Universal Robots PolyScope program: tcp_debug.urp

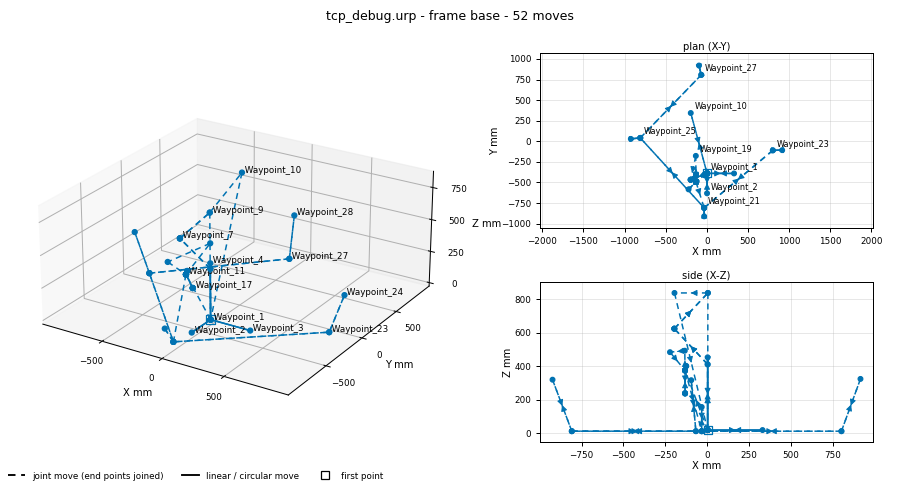
[picture p0: tool path of tcp_debug.urp in frame base, 52 of 52 moves have a stored position in this frame; points joined in program order, loops and branches not executed]
Program tcp_debug (installation=default directory=/programs/robviz createdIn=5.13.0 lastSavedIn=5.13.0 robotSerialNumber=20185501065)
Calibrated DH parameters: a=[0.000073, -0.261994, -0.164879, -0.000046, 0.000172, 0]; d=[0.162442, 111.219294, -268.471343, 157.385991, 0.099874, 0.099634]; alpha=[1.569873, -0.003012, -0.002263, 1.572206, -1.569596, 0]; deltaTheta=[0, -0.907061, 8.327173, -1.13692, -0.000001, 0]
InitVariablesNode
Robot Program (runOnlyOnce=false)
  Folder axis_aligned
    MoveL speed 250 mm/s, acceleration 1200 mm/s^2 (useActiveTCP=true) feature=Base
      Waypoint Waypoint_1: TCP in base x=2.814 y=-389.968 z=17.766 mm, rx=-2.8853 ry=-1.2149 rz=-0.0022 rad; joints [-69.728, -101.525, -140.49, -28.688, 89.823, -205.228] deg; TCP offset x=0 y=0 z=113.6 mm, rx=0 ry=0 rz=0 rad
      Waypoint Waypoint_2: TCP in base x=2.821 y=-632.109 z=17.753 mm, rx=-2.8853 ry=-1.2148 rz=-0.0023 rad; joints [-77.585, -124.965, -100.202, -45.538, 89.728, -213.114] deg
      Waypoint Waypoint_1: TCP in base x=2.814 y=-389.968 z=17.766 mm, rx=-2.8853 ry=-1.2149 rz=-0.0022 rad; joints [-69.728, -101.525, -140.49, -28.688, 89.823, -205.228] deg
    MoveL speed 250 mm/s, acceleration 1200 mm/s^2 (useActiveTCP=true) feature=Base
      Waypoint Waypoint_4: TCP in base x=2.832 y=-389.973 z=452.14 mm, rx=-2.8852 ry=-1.2149 rz=-0.0022 rad; joints [-69.77, -74.724, -91.391, -104.589, 89.981, -205.093] deg
      Waypoint Waypoint_1: TCP in base x=2.814 y=-389.968 z=17.766 mm, rx=-2.8853 ry=-1.2149 rz=-0.0022 rad; joints [-69.728, -101.525, -140.49, -28.688, 89.823, -205.228] deg
    MoveL speed 250 mm/s, acceleration 1200 mm/s^2 (useActiveTCP=true) feature=Base
      Waypoint Waypoint_3: TCP in base x=330.658 y=-390.809 z=17.849 mm, rx=-2.8853 ry=-1.215 rz=-0.0022 rad; joints [-34.907, -113.489, -121.144, -35.922, 90.163, -170.43] deg
      Waypoint Waypoint_1: TCP in base x=2.814 y=-389.968 z=17.766 mm, rx=-2.8853 ry=-1.2149 rz=-0.0022 rad; joints [-69.728, -101.525, -140.49, -28.688, 89.823, -205.228] deg
    MoveL speed 250 mm/s, acceleration 1200 mm/s^2 (useActiveTCP=true) feature=Base
      Waypoint Waypoint_5: TCP in base x=2.809 y=-389.964 z=17.76 mm, rx=-3.1106 ry=0.3715 rz=-0.0104 rad; joints [-70.027, -101.578, -140.604, -28.169, 90.338, -146.242] deg
      Waypoint Waypoint_1: TCP in base x=2.814 y=-389.968 z=17.766 mm, rx=-2.8853 ry=-1.2149 rz=-0.0022 rad; joints [-69.728, -101.525, -140.49, -28.688, 89.823, -205.228] deg
    MoveJ speed 60 deg/s, acceleration 80 deg/s^2 (useActiveTCP=true) feature=Base
      Waypoint Waypoint_6: TCP in base x=2.818 y=-389.957 z=410.089 mm, rx=-2.8853 ry=-1.2149 rz=-0.0022 rad; joints [-69.781, -73.648, -98.399, -98.655, 89.97, -205.104] deg
      Waypoint Waypoint_7: TCP in base x=-195.933 y=-467.312 z=623.185 mm, rx=-2.0027 ry=-0.8591 rz=2.1736 rad; joints [-69.778, -73.646, -98.397, -98.654, 0.001, -205.104] deg
      Waypoint Waypoint_8: TCP in base x=-195.946 y=-467.308 z=623.168 mm, rx=2.0294 ry=0.3823 rz=-2.0309 rad; joints [-69.78, -73.646, -98.399, -98.658, -0.001, -180] deg
      Waypoint Waypoint_9: TCP in base x=4.451 y=-394.853 z=836.583 mm, rx=-0.0013 ry=0.0189 rz=-2.7826 rad; joints [-69.782, -73.645, -98.395, -98.653, -90.001, -179.996] deg
      Waypoint Waypoint_1: TCP in base x=2.814 y=-389.968 z=17.766 mm, rx=-2.8853 ry=-1.2149 rz=-0.0022 rad; joints [-69.728, -101.525, -140.49, -28.688, 89.823, -205.228] deg
    MoveJ speed 60 deg/s, acceleration 80 deg/s^2 (useActiveTCP=true) feature=Base
      Waypoint Waypoint_6: TCP in base x=2.818 y=-389.957 z=410.089 mm, rx=-2.8853 ry=-1.2149 rz=-0.0022 rad; joints [-69.781, -73.648, -98.399, -98.655, 89.97, -205.104] deg
      Waypoint Waypoint_7: TCP in base x=-195.933 y=-467.312 z=623.185 mm, rx=-2.0027 ry=-0.8591 rz=2.1736 rad; joints [-69.778, -73.646, -98.397, -98.654, 0.001, -205.104] deg
      Waypoint Waypoint_8: TCP in base x=-195.946 y=-467.308 z=623.168 mm, rx=2.0294 ry=0.3823 rz=-2.0309 rad; joints [-69.78, -73.646, -98.399, -98.658, -0.001, -180] deg
      Waypoint Waypoint_9: TCP in base x=4.451 y=-394.853 z=836.583 mm, rx=-0.0013 ry=0.0189 rz=-2.7826 rad; joints [-69.782, -73.645, -98.395, -98.653, -90.001, -179.996] deg
      Waypoint Waypoint_10: TCP in base x=-195.137 y=343.292 z=836.575 mm, rx=-0.0131 ry=-0.0043 rz=0.8645 rad; joints [-220.812, -73.644, -98.397, -98.653, -90, -180] deg
      Waypoint Waypoint_1: TCP in base x=2.814 y=-389.968 z=17.766 mm, rx=-2.8853 ry=-1.2149 rz=-0.0022 rad; joints [-69.728, -101.525, -140.49, -28.688, 89.823, -205.228] deg
  Folder Joint_aligned
    MoveJ speed 60 deg/s, acceleration 80 deg/s^2 (useActiveTCP=true) feature=Base
      Waypoint Waypoint_11: TCP in base x=-132.053 y=-492.907 z=374.127 mm, rx=3.1404 ry=0.0085 rz=0.0037 rad; joints [-89.999, -89.996, -90.003, -90, 89.996, -180.004] deg
    MoveJ speed 60 deg/s, acceleration 80 deg/s^2 (useActiveTCP=true) feature=Base
      Waypoint Waypoint_13: TCP in base x=-132.026 y=-492.922 z=374.146 mm, rx=-2.6575 ry=-0.0064 rz=-0.0049 rad; joints [-89.964, -105.384, -69.147, -123.273, 90.108, -179.962] deg
      Waypoint Waypoint_11: TCP in base x=-132.053 y=-492.907 z=374.127 mm, rx=3.1404 ry=0.0085 rz=0.0037 rad; joints [-89.999, -89.996, -90.003, -90, 89.996, -180.004] deg
    MoveJ speed 60 deg/s, acceleration 80 deg/s^2 (useActiveTCP=true) feature=Base
      Waypoint Waypoint_12: TCP in base x=-132.029 y=-492.937 z=374.113 mm, rx=2.2136 ry=2.2256 rz=0.0013 rad; joints [-89.998, -90, -90.001, -89.999, 90, -270.003] deg
      Waypoint Waypoint_11: TCP in base x=-132.053 y=-492.907 z=374.127 mm, rx=3.1404 ry=0.0085 rz=0.0037 rad; joints [-89.999, -89.996, -90.003, -90, 89.996, -180.004] deg
    MoveL speed 250 mm/s, acceleration 1200 mm/s^2 (useActiveTCP=true) feature=Base
      Waypoint Waypoint_16: TCP in base x=-125.14 y=-487.309 z=399.99 mm, rx=3.1404 ry=0.0083 rz=0.0036 rad; joints [-89.182, -89.109, -87.104, -93.788, 90.004, -179.174] deg
      Waypoint Waypoint_14: TCP in base x=-125.124 y=-487.317 z=399.994 mm, rx=0.005 ry=0.0018 rz=-3.1364 rad; joints [-89.047, -118.699, -123.868, -27.427, -90.062, -180.769] deg
      Waypoint Waypoint_11: TCP in base x=-132.053 y=-492.907 z=374.127 mm, rx=3.1404 ry=0.0085 rz=0.0037 rad; joints [-89.999, -89.996, -90.003, -90, 89.996, -180.004] deg
    MoveL speed 250 mm/s, acceleration 1200 mm/s^2 (useActiveTCP=true) feature=Base
      Waypoint Waypoint_17: TCP in base x=-131.904 y=-409.398 z=236.983 mm, rx=3.1404 ry=0.0086 rz=0.0032 rad; joints [-89.998, -81.84, -117.949, -70.211, 89.957, -180.013] deg
      Waypoint Waypoint_15: TCP in base x=-131.907 y=-409.399 z=236.983 mm, rx=-1.5227 ry=-0.0025 rz=-0.0059 rad; joints [-89.932, -129.496, -75.161, -158.166, 90.275, -180.017] deg
      Waypoint Waypoint_17: TCP in base x=-131.904 y=-409.398 z=236.983 mm, rx=3.1404 ry=0.0086 rz=0.0032 rad; joints [-89.998, -81.84, -117.949, -70.211, 89.957, -180.013] deg
      Waypoint Waypoint_18: TCP in base x=-131.896 y=-409.385 z=236.971 mm, rx=2.7868 ry=0.0068 rz=1.4425 rad; joints [-111.778, -97.386, -109.544, -90.401, 139.249, -214.518] deg
      Waypoint Waypoint_17: TCP in base x=-131.904 y=-409.398 z=236.983 mm, rx=3.1404 ry=0.0086 rz=0.0032 rad; joints [-89.998, -81.84, -117.949, -70.211, 89.957, -180.013] deg
    MoveJ speed 60 deg/s, acceleration 80 deg/s^2 (useActiveTCP=true) feature=Base
      Waypoint Waypoint_11: TCP in base x=-132.053 y=-492.907 z=374.127 mm, rx=3.1404 ry=0.0085 rz=0.0037 rad; joints [-89.999, -89.996, -90.003, -90, 89.996, -180.004] deg
      Waypoint Waypoint_19: TCP in base x=-133.583 y=-177.458 z=491.729 mm, rx=-1.5512 ry=-0.0062 rz=0.0002 rad; joints [-89.998, -89.995, -90.003, -181.192, 89.993, -180.004] deg
      Waypoint Waypoint_20: TCP in base x=-221.952 y=-584.173 z=482.94 mm, rx=-0.4357 ry=-2.0039 rz=1.9587 rad; joints [-89.998, -89.995, -90.003, -181.194, -64.933, -180.002] deg
      Waypoint Waypoint_11: TCP in base x=-132.053 y=-492.907 z=374.127 mm, rx=3.1404 ry=0.0085 rz=0.0037 rad; joints [-89.999, -89.996, -90.003, -90, 89.996, -180.004] deg
  Folder Extremes
    MoveJ speed 60 deg/s, acceleration 80 deg/s^2 (useActiveTCP=true) feature=Base
      Waypoint Waypoint_21: TCP in base x=-32.534 y=-808.646 z=11.061 mm, rx=3.1403 ry=0.0084 rz=0.0037 rad; joints [-82.824, -145.256, -62.064, -62.663, 89.912, -173.021] deg
      Waypoint Waypoint_22: TCP in base x=-32.515 y=-912.045 z=155.569 mm, rx=1.558 ry=0.006 rz=-0.0025 rad; joints [-81.635, -158.812, -63.233, 42.733, 81.808, -180.542] deg
      Waypoint Waypoint_21: TCP in base x=-32.534 y=-808.646 z=11.061 mm, rx=3.1403 ry=0.0084 rz=0.0037 rad; joints [-82.824, -145.256, -62.064, -62.663, 89.912, -173.021] deg
    MoveJ speed 60 deg/s, acceleration 80 deg/s^2 (useActiveTCP=true) feature=Base
      Waypoint Waypoint_23: TCP in base x=801.766 y=-110.113 z=11.048 mm, rx=-2.3196 ry=-2.1176 rz=-0.0041 rad; joints [1.659, -145.256, -62.064, -62.663, 89.914, -173.02] deg
      Waypoint Waypoint_24: TCP in base x=915.405 y=-107.936 z=323.23 mm, rx=1.2916 ry=1.173 rz=1.318 rad; joints [1.66, -145.256, -62.063, 26.994, 89.91, -173.021] deg
      Waypoint Waypoint_23: TCP in base x=801.766 y=-110.113 z=11.048 mm, rx=-2.3196 ry=-2.1176 rz=-0.0041 rad; joints [1.659, -145.256, -62.064, -62.663, 89.914, -173.02] deg
      Waypoint Waypoint_21: TCP in base x=-32.534 y=-808.646 z=11.061 mm, rx=3.1403 ry=0.0084 rz=0.0037 rad; joints [-82.824, -145.256, -62.064, -62.663, 89.912, -173.021] deg
    MoveJ speed 60 deg/s, acceleration 80 deg/s^2 (useActiveTCP=true) feature=Base
      Waypoint Waypoint_25: TCP in base x=-808.268 y=41.037 z=11.055 mm, rx=2.2138 ry=-2.2254 rz=0.0012 rad; joints [-173.427, -145.257, -62.063, -62.662, 89.912, -173.02] deg
      Waypoint Waypoint_26: TCP in base x=-923.314 y=28.875 z=318.694 mm, rx=1.1931 ry=-1.2055 rz=-1.0219 rad; joints [-173.427, -145.254, -62.063, 25.779, 89.914, -173.018] deg
      Waypoint Waypoint_25: TCP in base x=-808.268 y=41.037 z=11.055 mm, rx=2.2138 ry=-2.2254 rz=0.0012 rad; joints [-173.427, -145.257, -62.063, -62.662, 89.912, -173.02] deg
    MoveJ speed 60 deg/s, acceleration 80 deg/s^2 (useActiveTCP=true) feature=Base
      Waypoint Waypoint_27: TCP in base x=-67.316 y=806.506 z=11.067 mm, rx=0.202 ry=-3.1326 rz=-0.0018 rad; joints [-255.749, -145.256, -62.063, -62.661, 89.912, -173.018] deg
      Waypoint Waypoint_28: TCP in base x=-95.06 y=920.192 z=315.585 mm, rx=0.1297 ry=-2.0935 rz=-1.9804 rad; joints [-255.751, -145.255, -62.062, 24.954, 89.914, -173.021] deg
      Waypoint Waypoint_27: TCP in base x=-67.316 y=806.506 z=11.067 mm, rx=0.202 ry=-3.1326 rz=-0.0018 rad; joints [-255.749, -145.256, -62.063, -62.661, 89.912, -173.018] deg
      Waypoint Waypoint_25: TCP in base x=-808.268 y=41.037 z=11.055 mm, rx=2.2138 ry=-2.2254 rz=0.0012 rad; joints [-173.427, -145.257, -62.063, -62.662, 89.912, -173.02] deg
      Waypoint Waypoint_21: TCP in base x=-32.534 y=-808.646 z=11.061 mm, rx=3.1403 ry=0.0084 rz=0.0037 rad; joints [-82.824, -145.256, -62.064, -62.663, 89.912, -173.021] deg
